// TIA Portal V18 export
// export: Created 2026-06-06T00:00:00Z, ExportSetting WithDefaults
VAR_GLOBAL   // PLC tag table "AI_Tags"
   AI_Nut_Khoi_Dong AT %I0.0 : Bool;   // Nút khởi động vật lý
   AI_Nut_Khoi_Dong_HMI AT %M110.0 : Bool;   // Tín hiệu mô phỏng/HMI song song cho Nút khởi động vật lý
   AI_Nut_Khoi_Dong_HMI_Gated AT %M320.0 : Bool;   // Tín hiệu HMI đã qua xử lý chế độ cho Nút khởi động vật lý
   AI_Nut_Khoi_Dong_Eff AT %M320.1 : Bool;   // Tín hiệu thực tế/mô phỏng hiệu dụng cho Nút khởi động vật lý
   AI_Nut_Dung AT %I0.1 : Bool;   // Nút dừng vật lý
   AI_Nut_Dung_HMI AT %M110.1 : Bool;   // Tín hiệu mô phỏng/HMI song song cho Nút dừng vật lý
   AI_Nut_Dung_HMI_Gated AT %M320.2 : Bool;   // Tín hiệu HMI đã qua xử lý chế độ cho Nút dừng vật lý
   AI_Nut_Dung_Eff AT %M320.3 : Bool;   // Tín hiệu thực tế/mô phỏng hiệu dụng cho Nút dừng vật lý
   AI_Nut_Reset AT %I0.2 : Bool;   // Nút reset lỗi vật lý
   AI_Nut_Reset_HMI AT %M110.2 : Bool;   // Tín hiệu mô phỏng/HMI song song cho Nút reset lỗi vật lý
   AI_Nut_Reset_HMI_Gated AT %M320.4 : Bool;   // Tín hiệu HMI đã qua xử lý chế độ cho Nút reset lỗi vật lý
   AI_Nut_Reset_Eff AT %M320.5 : Bool;   // Tín hiệu thực tế/mô phỏng hiệu dụng cho Nút reset lỗi vật lý
   AI_Nut_EStop AT %I0.3 : Bool;   // Nút dừng khẩn vật lý
   AI_Nut_EStop_HMI AT %M110.3 : Bool;   // Tín hiệu mô phỏng/HMI song song cho Nút dừng khẩn vật lý
   AI_Nut_EStop_HMI_Gated AT %M320.6 : Bool;   // Tín hiệu HMI đã qua xử lý chế độ cho Nút dừng khẩn vật lý
   AI_Nut_EStop_Eff AT %M320.7 : Bool;   // Tín hiệu thực tế/mô phỏng hiệu dụng cho Nút dừng khẩn vật lý
   AI_FT3200_Bon1 AT %ID100 : Real;   // Cảm biến lưu lượng nước dosing vào Bồn 1
   AI_FT3200_Bon1_HMI AT %MD700 : Real;   // Giá trị mô phỏng/HMI song song cho Cảm biến lưu lượng nước dosing vào Bồn 1
   AI_FT3200_Bon1_Use_HMI AT %M420.0 : Bool;   // Chọn chế độ mô phỏng HMI cho Cảm biến lưu lượng nước dosing vào Bồn 1
   AI_FT3200_Bon1_Sim_Req AT %M321.0 : Bool;   // Yêu cầu mô phỏng cảm biến cho Cảm biến lưu lượng nước dosing vào Bồn 1
   AI_FT3200_Bon1_Sim_Active AT %M321.1 : Bool;   // Mô phỏng cảm biến đang hoạt động cho Cảm biến lưu lượng nước dosing vào Bồn 1
   AI_FT3200_Bon1_Eff AT %MD704 : Real;   // Giá trị thực tế/mô phỏng hiệu dụng cho Cảm biến lưu lượng nước dosing vào Bồn 1
   AI_FQ3200_Bon1 AT %ID104 : Real;   // Bộ đếm lưu lượng tích lũy Bồn 1
   AI_FQ3200_Bon1_HMI AT %MD708 : Real;   // Giá trị mô phỏng/HMI song song cho Bộ đếm lưu lượng tích lũy Bồn 1
   AI_FQ3200_Bon1_Use_HMI AT %M420.1 : Bool;   // Chọn chế độ mô phỏng HMI cho Bộ đếm lưu lượng tích lũy Bồn 1
   AI_FQ3200_Bon1_Sim_Req AT %M321.2 : Bool;   // Yêu cầu mô phỏng cảm biến cho Bộ đếm lưu lượng tích lũy Bồn 1
   AI_FQ3200_Bon1_Sim_Active AT %M321.3 : Bool;   // Mô phỏng cảm biến đang hoạt động cho Bộ đếm lưu lượng tích lũy Bồn 1
   AI_FQ3200_Bon1_Eff AT %MD712 : Real;   // Giá trị thực tế/mô phỏng hiệu dụng cho Bộ đếm lưu lượng tích lũy Bồn 1
   AI_LS3202_Bon1_Cao AT %I0.4 : Bool;   // Cảm biến mức cao Bồn 1
   AI_LS3202_Bon1_Cao_HMI AT %M110.4 : Bool;   // Tín hiệu mô phỏng/HMI song song cho Cảm biến mức cao Bồn 1
   AI_LS3202_Bon1_Cao_HMI_Gated AT %M321.4 : Bool;   // Tín hiệu HMI đã qua xử lý chế độ cho Cảm biến mức cao Bồn 1
   AI_LS3202_Bon1_Cao_Eff AT %M321.5 : Bool;   // Tín hiệu thực tế/mô phỏng hiệu dụng cho Cảm biến mức cao Bồn 1
   AI_LT3203_Bon1 AT %ID108 : Real;   // Cảm biến mức liên tục Bồn 1
   AI_LT3203_Bon1_HMI AT %MD716 : Real;   // Giá trị mô phỏng/HMI song song cho Cảm biến mức liên tục Bồn 1
   AI_LT3203_Bon1_Use_HMI AT %M420.2 : Bool;   // Chọn chế độ mô phỏng HMI cho Cảm biến mức liên tục Bồn 1
   AI_LT3203_Bon1_Sim_Req AT %M321.6 : Bool;   // Yêu cầu mô phỏng cảm biến cho Cảm biến mức liên tục Bồn 1
   AI_LT3203_Bon1_Sim_Active AT %M321.7 : Bool;   // Mô phỏng cảm biến đang hoạt động cho Cảm biến mức liên tục Bồn 1
   AI_LT3203_Bon1_Eff AT %MD720 : Real;   // Giá trị thực tế/mô phỏng hiệu dụng cho Cảm biến mức liên tục Bồn 1
   AI_TT3204_Bon1 AT %ID112 : Real;   // Cảm biến nhiệt độ Bồn 1
   AI_TT3204_Bon1_HMI AT %MD724 : Real;   // Giá trị mô phỏng/HMI song song cho Cảm biến nhiệt độ Bồn 1
   AI_TT3204_Bon1_Use_HMI AT %M420.3 : Bool;   // Chọn chế độ mô phỏng HMI cho Cảm biến nhiệt độ Bồn 1
   AI_TT3204_Bon1_Sim_Req AT %M322.0 : Bool;   // Yêu cầu mô phỏng cảm biến cho Cảm biến nhiệt độ Bồn 1
   AI_TT3204_Bon1_Sim_Active AT %M322.1 : Bool;   // Mô phỏng cảm biến đang hoạt động cho Cảm biến nhiệt độ Bồn 1
   AI_TT3204_Bon1_Eff AT %MD728 : Real;   // Giá trị thực tế/mô phỏng hiệu dụng cho Cảm biến nhiệt độ Bồn 1
   AI_FT3205_Bon2 AT %ID116 : Real;   // Cảm biến lưu lượng nước dosing vào Bồn 2
   AI_FT3205_Bon2_HMI AT %MD732 : Real;   // Giá trị mô phỏng/HMI song song cho Cảm biến lưu lượng nước dosing vào Bồn 2
   AI_FT3205_Bon2_Use_HMI AT %M420.4 : Bool;   // Chọn chế độ mô phỏng HMI cho Cảm biến lưu lượng nước dosing vào Bồn 2
   AI_FT3205_Bon2_Sim_Req AT %M322.2 : Bool;   // Yêu cầu mô phỏng cảm biến cho Cảm biến lưu lượng nước dosing vào Bồn 2
   AI_FT3205_Bon2_Sim_Active AT %M322.3 : Bool;   // Mô phỏng cảm biến đang hoạt động cho Cảm biến lưu lượng nước dosing vào Bồn 2
   AI_FT3205_Bon2_Eff AT %MD736 : Real;   // Giá trị thực tế/mô phỏng hiệu dụng cho Cảm biến lưu lượng nước dosing vào Bồn 2
   AI_FQ3205_Bon2 AT %ID120 : Real;   // Bộ đếm lưu lượng tích lũy Bồn 2
   AI_FQ3205_Bon2_HMI AT %MD740 : Real;   // Giá trị mô phỏng/HMI song song cho Bộ đếm lưu lượng tích lũy Bồn 2
   AI_FQ3205_Bon2_Use_HMI AT %M420.5 : Bool;   // Chọn chế độ mô phỏng HMI cho Bộ đếm lưu lượng tích lũy Bồn 2
   AI_FQ3205_Bon2_Sim_Req AT %M322.4 : Bool;   // Yêu cầu mô phỏng cảm biến cho Bộ đếm lưu lượng tích lũy Bồn 2
   AI_FQ3205_Bon2_Sim_Active AT %M322.5 : Bool;   // Mô phỏng cảm biến đang hoạt động cho Bộ đếm lưu lượng tích lũy Bồn 2
   AI_FQ3205_Bon2_Eff AT %MD744 : Real;   // Giá trị thực tế/mô phỏng hiệu dụng cho Bộ đếm lưu lượng tích lũy Bồn 2
   AI_LT3209_Bon2 AT %ID124 : Real;   // Cảm biến mức liên tục Bồn 2
   AI_LT3209_Bon2_HMI AT %MD748 : Real;   // Giá trị mô phỏng/HMI song song cho Cảm biến mức liên tục Bồn 2
   AI_LT3209_Bon2_Use_HMI AT %M420.6 : Bool;   // Chọn chế độ mô phỏng HMI cho Cảm biến mức liên tục Bồn 2
   AI_LT3209_Bon2_Sim_Req AT %M322.6 : Bool;   // Yêu cầu mô phỏng cảm biến cho Cảm biến mức liên tục Bồn 2
   AI_LT3209_Bon2_Sim_Active AT %M322.7 : Bool;   // Mô phỏng cảm biến đang hoạt động cho Cảm biến mức liên tục Bồn 2
   AI_LT3209_Bon2_Eff AT %MD752 : Real;   // Giá trị thực tế/mô phỏng hiệu dụng cho Cảm biến mức liên tục Bồn 2
   AI_TT3208_Bon2 AT %ID128 : Real;   // Cảm biến nhiệt độ Bồn 2
   AI_TT3208_Bon2_HMI AT %MD756 : Real;   // Giá trị mô phỏng/HMI song song cho Cảm biến nhiệt độ Bồn 2
   AI_TT3208_Bon2_Use_HMI AT %M420.7 : Bool;   // Chọn chế độ mô phỏng HMI cho Cảm biến nhiệt độ Bồn 2
   AI_TT3208_Bon2_Sim_Req AT %M323.0 : Bool;   // Yêu cầu mô phỏng cảm biến cho Cảm biến nhiệt độ Bồn 2
   AI_TT3208_Bon2_Sim_Active AT %M323.1 : Bool;   // Mô phỏng cảm biến đang hoạt động cho Cảm biến nhiệt độ Bồn 2
   AI_TT3208_Bon2_Eff AT %MD760 : Real;   // Giá trị thực tế/mô phỏng hiệu dụng cho Cảm biến nhiệt độ Bồn 2
   AI_V3230_Nuoc_Bon1 AT %Q0.0 : Bool;   // Van on/off cấp nước Bồn 1
   AI_V3230_Nuoc_Bon1_M AT %M220.0 : Bool;   // Tag gương phản hồi HMI cho Van on/off cấp nước Bồn 1
   AI_CV3201_Nuoc_Bon1 AT %QD100 : Real;   // Van tuyến tính cấp nước Bồn 1
   AI_CV3201_Nuoc_Bon1_M AT %MD1200 : Real;   // Tag gương phản hồi HMI cho Van tuyến tính cấp nước Bồn 1
   AI_AGTR3260_Khuay_Bon1 AT %Q0.1 : Bool;   // Động cơ khuấy Bồn 1
   AI_AGTR3260_Khuay_Bon1_M AT %M220.1 : Bool;   // Tag gương phản hồi HMI cho Động cơ khuấy Bồn 1
   AI_AGTR3260_Toc_Do_AO AT %QD104 : Real;   // Tín hiệu tốc độ khuấy Bồn 1
   AI_AGTR3260_Toc_Do_AO_M AT %MD1204 : Real;   // Tag gương phản hồi HMI cho Tín hiệu tốc độ khuấy Bồn 1
   AI_V3232_Xa_Bon1 AT %Q0.2 : Bool;   // Van xả đáy Bồn 1 số 1
   AI_V3232_Xa_Bon1_M AT %M220.2 : Bool;   // Tag gương phản hồi HMI cho Van xả đáy Bồn 1 số 1
   AI_V3233_Xa_Bon1 AT %Q0.3 : Bool;   // Van xả đáy Bồn 1 số 2
   AI_V3233_Xa_Bon1_M AT %M220.3 : Bool;   // Tag gương phản hồi HMI cho Van xả đáy Bồn 1 số 2
   AI_V3234_Xa_Bon1 AT %Q0.4 : Bool;   // Van xả đáy Bồn 1 số 3
   AI_V3234_Xa_Bon1_M AT %M220.4 : Bool;   // Tag gương phản hồi HMI cho Van xả đáy Bồn 1 số 3
   AI_V3235_Nuoc_Bon2 AT %Q0.5 : Bool;   // Van on/off cấp nước Bồn 2
   AI_V3235_Nuoc_Bon2_M AT %M220.5 : Bool;   // Tag gương phản hồi HMI cho Van on/off cấp nước Bồn 2
   AI_CV3206_Hoi_Bon2 AT %QD108 : Real;   // Van hơi/nhiệt Bồn 2 ở chế độ cho phép
   AI_CV3206_Hoi_Bon2_M AT %MD1208 : Real;   // Tag gương phản hồi HMI cho Van hơi/nhiệt Bồn 2 ở chế độ cho phép
   AI_VFD_Bon2_Run AT %Q0.6 : Bool;   // Lệnh chạy VFD động cơ Bồn 2
   AI_VFD_Bon2_Run_M AT %M220.6 : Bool;   // Tag gương phản hồi HMI cho Lệnh chạy VFD động cơ Bồn 2
   AI_VFD_Bon2_Dao_Chieu AT %Q0.7 : Bool;   // Lệnh đảo chiều VFD động cơ Bồn 2
   AI_VFD_Bon2_Dao_Chieu_M AT %M220.7 : Bool;   // Tag gương phản hồi HMI cho Lệnh đảo chiều VFD động cơ Bồn 2
   AI_VFD_Bon2_Toc_Do_AO AT %QD112 : Real;   // Tốc độ đặt VFD Bồn 2 từ HMI setpoint
   AI_VFD_Bon2_Toc_Do_AO_M AT %MD1212 : Real;   // Tag gương phản hồi HMI cho Tốc độ đặt VFD Bồn 2 từ HMI setpoint
   AI_V3237_Xa_Bon2 AT %Q1.0 : Bool;   // Van xả đáy Bồn 2 số 1
   AI_V3237_Xa_Bon2_M AT %M221.0 : Bool;   // Tag gương phản hồi HMI cho Van xả đáy Bồn 2 số 1
   AI_V3238_Xa_Bon2 AT %Q1.1 : Bool;   // Van xả đáy Bồn 2 số 2
   AI_V3238_Xa_Bon2_M AT %M221.1 : Bool;   // Tag gương phản hồi HMI cho Van xả đáy Bồn 2 số 2
   AI_V3239_Xa_Bon2 AT %Q1.2 : Bool;   // Van xả đáy Bồn 2 số 3
   AI_V3239_Xa_Bon2_M AT %M221.2 : Bool;   // Tag gương phản hồi HMI cho Van xả đáy Bồn 2 số 3
   AI_Pump3264_Chuyen_Nhanh1 AT %Q1.3 : Bool;   // Bơm chuyển dung dịch Nhánh 1 xuống bồn chứa
   AI_Pump3264_Chuyen_Nhanh1_M AT %M221.3 : Bool;   // Tag gương phản hồi HMI cho Bơm chuyển dung dịch Nhánh 1 xuống bồn chứa
   AI_LT3302_BonChua1 AT %ID164 : Real;   // Cảm biến mức liên tục Bồn chứa 01
   AI_LT3302_BonChua1_HMI AT %MD828 : Real;   // Giá trị mô phỏng/HMI song song cho Cảm biến mức liên tục Bồn chứa 01
   AI_LT3302_BonChua1_Use_HMI AT %M422.0 : Bool;   // Chọn chế độ mô phỏng HMI cho Cảm biến mức liên tục Bồn chứa 01
   AI_LT3302_BonChua1_Sim_Req AT %M325.4 : Bool;   // Yêu cầu mô phỏng cảm biến cho Cảm biến mức liên tục Bồn chứa 01
   AI_LT3302_BonChua1_Sim_Active AT %M325.5 : Bool;   // Mô phỏng cảm biến đang hoạt động cho Cảm biến mức liên tục Bồn chứa 01
   AI_LT3302_BonChua1_Eff AT %MD832 : Real;   // Giá trị thực tế/mô phỏng hiệu dụng cho Cảm biến mức liên tục Bồn chứa 01
   AI_TT3301_BonChua1 AT %ID168 : Real;   // Cảm biến nhiệt độ Bồn chứa 01
   AI_TT3301_BonChua1_HMI AT %MD836 : Real;   // Giá trị mô phỏng/HMI song song cho Cảm biến nhiệt độ Bồn chứa 01
   AI_TT3301_BonChua1_Use_HMI AT %M422.1 : Bool;   // Chọn chế độ mô phỏng HMI cho Cảm biến nhiệt độ Bồn chứa 01
   AI_TT3301_BonChua1_Sim_Req AT %M325.6 : Bool;   // Yêu cầu mô phỏng cảm biến cho Cảm biến nhiệt độ Bồn chứa 01
   AI_TT3301_BonChua1_Sim_Active AT %M325.7 : Bool;   // Mô phỏng cảm biến đang hoạt động cho Cảm biến nhiệt độ Bồn chứa 01
   AI_TT3301_BonChua1_Eff AT %MD840 : Real;   // Giá trị thực tế/mô phỏng hiệu dụng cho Cảm biến nhiệt độ Bồn chứa 01
   AI_TT3303_TraoDoiNhiet AT %ID172 : Real;   // Cảm biến nhiệt độ bộ trao đổi nhiệt
   AI_TT3303_TraoDoiNhiet_HMI AT %MD844 : Real;   // Giá trị mô phỏng/HMI song song cho Cảm biến nhiệt độ bộ trao đổi nhiệt
   AI_TT3303_TraoDoiNhiet_Use_HMI AT %M422.2 : Bool;   // Chọn chế độ mô phỏng HMI cho Cảm biến nhiệt độ bộ trao đổi nhiệt
   AI_TT3303_TraoDoiNhiet_Sim_Req AT %M326.0 : Bool;   // Yêu cầu mô phỏng cảm biến cho Cảm biến nhiệt độ bộ trao đổi nhiệt
   AI_TT3303_TraoDoiNhiet_Sim_Active AT %M326.1 : Bool;   // Mô phỏng cảm biến đang hoạt động cho Cảm biến nhiệt độ bộ trao đổi nhiệt
   AI_TT3303_TraoDoiNhiet_Eff AT %MD848 : Real;   // Giá trị thực tế/mô phỏng hiệu dụng cho Cảm biến nhiệt độ bộ trao đổi nhiệt
   AI_LT3307_BonChua2 AT %ID176 : Real;   // Cảm biến mức liên tục Bồn chứa 02
   AI_LT3307_BonChua2_HMI AT %MD852 : Real;   // Giá trị mô phỏng/HMI song song cho Cảm biến mức liên tục Bồn chứa 02
   AI_LT3307_BonChua2_Use_HMI AT %M422.3 : Bool;   // Chọn chế độ mô phỏng HMI cho Cảm biến mức liên tục Bồn chứa 02
   AI_LT3307_BonChua2_Sim_Req AT %M326.2 : Bool;   // Yêu cầu mô phỏng cảm biến cho Cảm biến mức liên tục Bồn chứa 02
   AI_LT3307_BonChua2_Sim_Active AT %M326.3 : Bool;   // Mô phỏng cảm biến đang hoạt động cho Cảm biến mức liên tục Bồn chứa 02
   AI_LT3307_BonChua2_Eff AT %MD856 : Real;   // Giá trị thực tế/mô phỏng hiệu dụng cho Cảm biến mức liên tục Bồn chứa 02
   AI_TT3306_BonChua2 AT %ID180 : Real;   // Cảm biến nhiệt độ Bồn chứa 02
   AI_TT3306_BonChua2_HMI AT %MD860 : Real;   // Giá trị mô phỏng/HMI song song cho Cảm biến nhiệt độ Bồn chứa 02
   AI_TT3306_BonChua2_Use_HMI AT %M422.4 : Bool;   // Chọn chế độ mô phỏng HMI cho Cảm biến nhiệt độ Bồn chứa 02
   AI_TT3306_BonChua2_Sim_Req AT %M326.4 : Bool;   // Yêu cầu mô phỏng cảm biến cho Cảm biến nhiệt độ Bồn chứa 02
   AI_TT3306_BonChua2_Sim_Active AT %M326.5 : Bool;   // Mô phỏng cảm biến đang hoạt động cho Cảm biến nhiệt độ Bồn chứa 02
   AI_TT3306_BonChua2_Eff AT %MD864 : Real;   // Giá trị thực tế/mô phỏng hiệu dụng cho Cảm biến nhiệt độ Bồn chứa 02
   AI_PI3308_Truoc_Filter AT %ID184 : Real;   // Cảm biến áp suất trước màng lọc
   AI_PI3308_Truoc_Filter_HMI AT %MD868 : Real;   // Giá trị mô phỏng/HMI song song cho Cảm biến áp suất trước màng lọc
   AI_PI3308_Truoc_Filter_Use_HMI AT %M422.5 : Bool;   // Chọn chế độ mô phỏng HMI cho Cảm biến áp suất trước màng lọc
   AI_PI3308_Truoc_Filter_Sim_Req AT %M326.6 : Bool;   // Yêu cầu mô phỏng cảm biến cho Cảm biến áp suất trước màng lọc
   AI_PI3308_Truoc_Filter_Sim_Active AT %M326.7 : Bool;   // Mô phỏng cảm biến đang hoạt động cho Cảm biến áp suất trước màng lọc
   AI_PI3308_Truoc_Filter_Eff AT %MD872 : Real;   // Giá trị thực tế/mô phỏng hiệu dụng cho Cảm biến áp suất trước màng lọc
   AI_FT3309_Xa_Thanh_Pham AT %ID188 : Real;   // Cảm biến lưu lượng xả thành phẩm
   AI_FT3309_Xa_Thanh_Pham_HMI AT %MD876 : Real;   // Giá trị mô phỏng/HMI song song cho Cảm biến lưu lượng xả thành phẩm
   AI_FT3309_Xa_Thanh_Pham_Use_HMI AT %M422.6 : Bool;   // Chọn chế độ mô phỏng HMI cho Cảm biến lưu lượng xả thành phẩm
   AI_FT3309_Xa_Thanh_Pham_Sim_Req AT %M327.0 : Bool;   // Yêu cầu mô phỏng cảm biến cho Cảm biến lưu lượng xả thành phẩm
   AI_FT3309_Xa_Thanh_Pham_Sim_Active AT %M327.1 : Bool;   // Mô phỏng cảm biến đang hoạt động cho Cảm biến lưu lượng xả thành phẩm
   AI_FT3309_Xa_Thanh_Pham_Eff AT %MD880 : Real;   // Giá trị thực tế/mô phỏng hiệu dụng cho Cảm biến lưu lượng xả thành phẩm
   AI_LSH3310_Pheu_Cao AT %I0.6 : Bool;   // Cảm biến mức cao phễu chiết rót
   AI_LSH3310_Pheu_Cao_HMI AT %M110.6 : Bool;   // Tín hiệu mô phỏng/HMI song song cho Cảm biến mức cao phễu chiết rót
   AI_LSH3310_Pheu_Cao_HMI_Gated AT %M327.2 : Bool;   // Tín hiệu HMI đã qua xử lý chế độ cho Cảm biến mức cao phễu chiết rót
   AI_LSH3310_Pheu_Cao_Eff AT %M327.3 : Bool;   // Tín hiệu thực tế/mô phỏng hiệu dụng cho Cảm biến mức cao phễu chiết rót
   AI_LSL3311_Pheu_Thap AT %I0.7 : Bool;   // Cảm biến mức thấp phễu chiết rót
   AI_LSL3311_Pheu_Thap_HMI AT %M110.7 : Bool;   // Tín hiệu mô phỏng/HMI song song cho Cảm biến mức thấp phễu chiết rót
   AI_LSL3311_Pheu_Thap_HMI_Gated AT %M327.4 : Bool;   // Tín hiệu HMI đã qua xử lý chế độ cho Cảm biến mức thấp phễu chiết rót
   AI_LSL3311_Pheu_Thap_Eff AT %M327.5 : Bool;   // Tín hiệu thực tế/mô phỏng hiệu dụng cho Cảm biến mức thấp phễu chiết rót
   AI_V3331_Xa_BonChua1 AT %Q3.0 : Bool;   // Van xả đáy Bồn chứa 01 số 1
   AI_V3331_Xa_BonChua1_M AT %M223.0 : Bool;   // Tag gương phản hồi HMI cho Van xả đáy Bồn chứa 01 số 1
   AI_V3332_Xa_BonChua1 AT %Q3.1 : Bool;   // Van xả đáy Bồn chứa 01 số 2
   AI_V3332_Xa_BonChua1_M AT %M223.1 : Bool;   // Tag gương phản hồi HMI cho Van xả đáy Bồn chứa 01 số 2
   AI_Pump3361_LuanChuyen_BonChua1 AT %Q3.2 : Bool;   // Bơm luân chuyển Bồn chứa 01
   AI_Pump3361_LuanChuyen_BonChua1_M AT %M223.2 : Bool;   // Tag gương phản hồi HMI cho Bơm luân chuyển Bồn chứa 01
   AI_Pump3362_Xa_BonChua1 AT %Q3.3 : Bool;   // Bơm xả Bồn chứa 01
   AI_Pump3362_Xa_BonChua1_M AT %M223.3 : Bool;   // Tag gương phản hồi HMI cho Bơm xả Bồn chứa 01
   AI_V3333_DieuHuong_BonChua1 AT %Q3.4 : Bool;   // Van điều hướng Bồn chứa 01 số 1
   AI_V3333_DieuHuong_BonChua1_M AT %M223.4 : Bool;   // Tag gương phản hồi HMI cho Van điều hướng Bồn chứa 01 số 1
   AI_V3334_DieuHuong_BonChua1 AT %Q3.5 : Bool;   // Van điều hướng Bồn chứa 01 số 2
   AI_V3334_DieuHuong_BonChua1_M AT %M223.5 : Bool;   // Tag gương phản hồi HMI cho Van điều hướng Bồn chứa 01 số 2
   AI_V3335_DieuHuong_BonChua1 AT %Q3.6 : Bool;   // Van điều hướng Bồn chứa 01 số 3
   AI_V3335_DieuHuong_BonChua1_M AT %M223.6 : Bool;   // Tag gương phản hồi HMI cho Van điều hướng Bồn chứa 01 số 3
   AI_CV3304_Nuoc_Lam_Mat AT %QD132 : Real;   // Van tuyến tính nước làm mát
   AI_CV3304_Nuoc_Lam_Mat_M AT %MD1232 : Real;   // Tag gương phản hồi HMI cho Van tuyến tính nước làm mát
   AI_V3338_Xa_BonChua2 AT %Q3.7 : Bool;   // Van xả đáy Bồn chứa 02 số 1
   AI_V3338_Xa_BonChua2_M AT %M223.7 : Bool;   // Tag gương phản hồi HMI cho Van xả đáy Bồn chứa 02 số 1
   AI_V3339_Xa_BonChua2 AT %Q4.0 : Bool;   // Van xả đáy Bồn chứa 02 số 2
   AI_V3339_Xa_BonChua2_M AT %M224.0 : Bool;   // Tag gương phản hồi HMI cho Van xả đáy Bồn chứa 02 số 2
   AI_Pump3364_Filter AT %Q4.1 : Bool;   // Bơm qua màng lọc CCP số 1
   AI_Pump3364_Filter_M AT %M224.1 : Bool;   // Tag gương phản hồi HMI cho Bơm qua màng lọc CCP số 1
   AI_Pump3365_Filter AT %Q4.2 : Bool;   // Bơm qua màng lọc CCP số 2
   AI_Pump3365_Filter_M AT %M224.2 : Bool;   // Tag gương phản hồi HMI cho Bơm qua màng lọc CCP số 2
   AI_V3340_Duong_Filter AT %Q4.3 : Bool;   // Van đường ống Filter số 1
   AI_V3340_Duong_Filter_M AT %M224.3 : Bool;   // Tag gương phản hồi HMI cho Van đường ống Filter số 1
   AI_V3341_Duong_Filter AT %Q4.4 : Bool;   // Van đường ống Filter số 2
   AI_V3341_Duong_Filter_M AT %M224.4 : Bool;   // Tag gương phản hồi HMI cho Van đường ống Filter số 2
   AI_CV_Filler_Cap_Dich AT %QD136 : Real;   // Van tuyến tính cấp dịch xuống phễu chiết rót
   AI_CV_Filler_Cap_Dich_M AT %MD1236 : Real;   // Tag gương phản hồi HMI cho Van tuyến tính cấp dịch xuống phễu chiết rót
   AI_Coi_Bao_Dong AT %Q4.5 : Bool;   // Còi báo động chung
   AI_Coi_Bao_Dong_M AT %M224.5 : Bool;   // Tag gương phản hồi HMI cho Còi báo động chung
   AI_HMI_Operator_Login AT %M422.7 : Bool;   // Đăng nhập quyền Operator
   AI_HMI_Engineer_Login AT %M423.0 : Bool;   // Đăng nhập quyền Engineer
   AI_HMI_Admin_Login AT %M423.1 : Bool;   // Đăng nhập quyền Admin
   AI_HMI_Che_Do_Manual AT %M423.2 : Bool;   // Cho phép điều khiển tay từng thiết bị
   AI_HMI_Ack_Alarm AT %M423.3 : Bool;   // Xác nhận cảnh báo
   AI_HMI_Reset_Alarm AT %M423.4 : Bool;   // Reset alarm bằng HMI
   AI_Gia_Lap_Mat_Ket_Noi_HMI AT %M423.5 : Bool;   // Nút giả lập mất kết nối PLC
   AI_HMI_User_Level AT %MW520 : Int;   // Mức quyền hiện tại: 1 Operator, 2 Engineer, 3 Admin
   AI_HMI_Cho_Phep_Sua_Thong_So AT %M327.6 : Bool;   // Cờ cho phép sửa công thức và PID
   AI_HMI_Alarm_Status AT %MW522 : Int;   // Mã cảnh báo tổng hợp cho WinCC TextList
   AI_HMI_AnToan_Status AT %MW524 : Int;   // Mã chẩn đoán an toàn ưu tiên
   AI_PLC1_Auto_Enable AT %M327.7 : Bool;   // Cho phép chạy Auto Nhánh 1 Bồn 1-2
   AI_PLC1_EStop_Latch AT %M328.0 : Bool;   // Chốt dừng khẩn HMI/SCADA Nhánh 1 Bồn 1-2
   AI_PLC1_Loi_Tong AT %M328.1 : Bool;   // Lỗi tổng khóa Auto Nhánh 1 Bồn 1-2
   AI_PLC1_Loi_Dry_Run AT %M328.2 : Bool;   // Lỗi chạy khô bơm Nhánh 1 Bồn 1-2
   AI_PLC1_Loi_Dosing AT %M328.3 : Bool;   // Lỗi quá thời gian dosing Nhánh 1 Bồn 1-2
   AI_PLC1_Loi_Truyen_Thong AT %M328.4 : Bool;   // Lỗi truyền thông mô phỏng Nhánh 1 Bồn 1-2
   AI_PLC1_State AT %MW526 : Int;   // Mã bước chu trình Nhánh 1 Bồn 1-2
   AI_PLC1_Step_Bon1_Dosing AT %M329.3 : Bool;   // Bồn 1 đang dosing nước
   AI_PLC1_Step_Bon1_Tip AT %M329.4 : Bool;   // Bồn 1 đang mô phỏng tip cốt tương Nhật Bản
   AI_PLC1_Step_Bon1_Khuay AT %M329.5 : Bool;   // Bồn 1 đang khuấy ban đầu
   AI_PLC1_Step_Bon1_Xa AT %M329.6 : Bool;   // Bồn 1 đang xả sang Bồn 2
   AI_PLC1_Step_Bon2_Dosing AT %M329.7 : Bool;   // Bồn 2 đang dosing bổ sung
   AI_PLC1_Step_Bon2_Tip AT %M330.0 : Bool;   // Bồn 2 đang tip phụ gia
   AI_PLC1_Step_Bon2_Khuay_Thuan AT %M330.1 : Bool;   // Bồn 2 khuấy chiều thuận
   AI_PLC1_Step_Bon2_Khuay_Nghich AT %M330.2 : Bool;   // Bồn 2 khuấy chiều ngược
   AI_PLC1_Step_Bon2_PID AT %M330.3 : Bool;   // Bồn 2 gia nhiệt PID
   AI_PLC1_Step_Bon2_Thanh_Trung AT %M330.4 : Bool;   // Bồn 2 giữ thời gian thanh trùng
   AI_PLC1_Me_Nhanh1_Hoan_Thanh AT %M330.5 : Bool;   // Nhánh 1 hoàn thành và sẵn sàng xả xuống bồn chứa
   AI_PLC1_Xa_Bon1_Xong AT %M330.6 : Bool;   // Bồn 1 đã xả hết
   AI_PLC1_Xa_Bon2_Xong AT %M330.7 : Bool;   // Bồn 2 đã xả hết
   AI_BonChua_Step_Nhan_Dich AT %M332.4 : Bool;   // Bồn chứa 01 đang nhận dịch từ nhánh hoàn thành
   AI_BonChua_Step_Giai_Nhiet AT %M332.5 : Bool;   // Bồn chứa 01 đang giải nhiệt xuống 45 độ C
   AI_BonChua_Step_Chuyen_Bon2 AT %M332.6 : Bool;   // Đang chuyển từ Bồn chứa 01 sang Bồn chứa 02
   AI_BonChua_Step_Loc_Chiet AT %M332.7 : Bool;   // Đang lọc CCP và chiết rót
   AI_BonChua_Me_Hoan_Thanh AT %M333.0 : Bool;   // Hoàn thành một mẻ sản xuất chung
   AI_BonChua_State AT %MW530 : Int;   // Mã bước cụm bồn chứa và lọc thành phẩm
   AI_BonChua_Owner_Nhanh1 AT %M333.1 : Bool;   // Mức ưu tiên Nhánh 1 sở hữu bồn chứa
   AI_BonChua_Owner_Nhanh2 AT %M333.2 : Bool;   // Mức ưu tiên Nhánh 2 sở hữu bồn chứa
   AI_PLC2_Me_Nhanh2_Hoan_Thanh_Nhan AT %M333.4 : Bool;   // Cờ PLC1 nhận trạng thái hoàn thành từ PLC2
   AI_PLC2_Me_Nhanh2_Hoan_Thanh_Nhan_HMI AT %M111.0 : Bool;   // Tín hiệu mô phỏng/HMI song song cho cờ PLC1 nhận trạng thái hoàn thành từ PLC2
   AI_PLC2_Xa_Bon4_Xong_Nhan AT %M333.5 : Bool;   // Cờ PLC1 nhận trạng thái xả xong Bồn 4 từ PLC2
   AI_Pump3265_Chuyen_Nhanh2_Cmd AT %M333.6 : Bool;   // Lệnh chạy bơm chuyển Nhánh 2 gửi sang PLC2
   AI_Pump3265_Chuyen_Nhanh2_Cmd_M AT %M224.7 : Bool;   // Tag gương phản hồi HMI cho lệnh chạy bơm chuyển Nhánh 2 gửi sang PLC2
   AI_PID_Bon4_SP_Recv AT %MD884 : Real;   // PID Bồn 4 Setpoint nhận từ PLC2
   AI_PID_Bon4_PV_Recv AT %MD888 : Real;   // PID Bồn 4 Process Value nhận từ PLC2
   AI_PID_Bon4_CV_Recv AT %MD892 : Real;   // PID Bồn 4 Control Value nhận từ PLC2
   AI_PLC2_State_Recv AT %MW532 : Int;   // Trạng thái hoạt động PLC2 nhận từ PLC2
   AI_PLC2_Loi_Tong_Recv AT %M334.0 : Bool;   // Cờ lỗi tổng PLC2 nhận từ PLC2
   AI_VFD_Bon2_iStep AT %MW60 : Int;   // Bước quét tuần tự Modbus VFD Bồn 2
   AI_VFD_Bon2_iStep_Reset AT %M335.5 : Bool;   // Cờ reset bộ đếm bước Modbus VFD Bồn 2
   AI_VFD_Bon2_Step0_Req AT %M335.6 : Bool;   // Yêu cầu bước 0 Modbus VFD Bồn 2
   AI_VFD_Bon2_Step1_Req AT %M335.7 : Bool;   // Yêu cầu bước 1 Modbus VFD Bồn 2
   AI_VFD_Bon2_Step2_Req AT %M336.0 : Bool;   // Yêu cầu bước 2 Modbus VFD Bồn 2
   AI_VFD_Bon2_Step3_Req AT %M336.1 : Bool;   // Yêu cầu bước 3 Modbus VFD Bồn 2
   AI_VFD_Bon2_MB_ControlWord AT %MW40 : Word;   // Control Word gửi VFD Bồn 2
   AI_VFD_Bon2_MB_FreqSetpoint AT %MW42 : Int;   // Frequency Setpoint gửi VFD Bồn 2
   AI_VFD_Bon2_MB_StatusWord AT %MW44 : Word;   // Status Word đọc từ VFD Bồn 2
   AI_VFD_Bon2_MB_ActualSpeed AT %MW46 : Int;   // Actual Speed đọc từ VFD Bồn 2
   AI_VFD_Bon2_MB_Error AT %M50.0 : Bool;   // Lỗi Modbus Master VFD Bồn 2
   AI_VFD_Bon2_MB_Busy AT %M50.1 : Bool;   // Modbus Master Busy VFD Bồn 2
   AI_VFD_Bon2_MB_Done AT %M50.2 : Bool;   // Modbus Master Done VFD Bồn 2
   AI_VFD_Bon2_MB_Status AT %MW52 : Word;   // Trạng thái Modbus Master VFD Bồn 2
   AI_VFD_Bon2_MBCL_Done AT %M51.0 : Bool;   // Modbus Comm Load Done VFD Bồn 2
   AI_VFD_Bon2_MBCL_Error AT %M51.1 : Bool;   // Modbus Comm Load Error VFD Bồn 2
   AI_VFD_Bon2_MBCL_Status AT %MW54 : Word;   // Trạng thái Modbus Comm Load VFD Bồn 2
   AI_VFD_Bon2_Freq_Temp AT %MD70 : Real;   // Biến tạm tần số VFD Bồn 2
   AI_VFD_Bon2_Actual_Speed_Feedback AT %MD74 : Real;   // Phản hồi tốc độ thực tế VFD Bồn 2
   AI_VFD_Bon2_Actual_Speed_Feedback_M AT %MD1240 : Real;   // Tag gương phản hồi HMI tốc độ thực tế VFD Bồn 2
   AI_Clock_1Hz AT %M100.5 : Bool;   // Clock 1Hz system memory bit
   AI_FirstScan AT %M101.0 : Bool;   // First Scan system memory bit
   AI_MB_TCP_iStep AT %MW80 : Int;   // Modbus TCP Client step
   AI_MB_TCP_REQ AT %M82.0 : Bool;   // Modbus TCP Client Request
   AI_MB_TCP_DONE AT %M82.2 : Bool;   // Modbus TCP Client Transaction Done
   AI_MB_TCP_ERROR AT %M82.3 : Bool;   // Modbus TCP Client Transaction Error
   AI_MB_TCP_BUSY AT %M82.6 : Bool;   // Modbus TCP Client Transaction Busy
   AI_MB_TCP_STATUS AT %MW84 : Word;   // Modbus TCP Client Status
   AI_MB_TCP_Mode AT %MB88 : USInt;   // Modbus TCP Client Mode
   AI_MB_TCP_DataAddr AT %MD90 : UDInt;   // Modbus TCP Client Data Address
   AI_MB_TCP_DataLen AT %MW94 : UInt;   // Modbus TCP Client Data Length
   AI_Nut_Khoi_Dong_Eff_Old AT %M83.0 : Bool;   // Old value of Start button
   AI_Nut_Khoi_Dong_Eff_Edge AT %M83.6 : Bool;   // Start command edge detected
   AI_Nut_Dung_Eff_Old AT %M83.1 : Bool;   // Old value of Stop button
   AI_Nut_Dung_Eff_Edge AT %M83.7 : Bool;   // Stop command edge detected
   AI_Nut_Reset_Eff_Old AT %M83.2 : Bool;   // Old value of Reset button
   AI_Nut_Reset_Eff_Edge AT %M84.0 : Bool;   // Reset command edge detected
   AI_Nut_EStop_Eff_Old AT %M83.3 : Bool;   // Old value of EStop button
   AI_Nut_EStop_Eff_Edge AT %M84.1 : Bool;   // EStop command edge detected
   AI_Pump3265_Chuyen_Nhanh2_Cmd_Old AT %M83.4 : Bool;   // Old value of Transfer command
   AI_Pump3265_Chuyen_Nhanh2_Cmd_Edge AT %M84.2 : Bool;   // Transfer command edge detected
   AI_PLC1_Load_Default_Cmd_Old AT %M83.5 : Bool;   // Old value of Load Recipe command
   AI_PLC1_Load_Default_Cmd_Edge AT %M84.3 : Bool;   // Load Recipe command edge detected
   AI_MB_TCP_Any_Cmd_Edge AT %M84.4 : Bool;   // Any handshake command edge detected
   AI_PLC1_Tip_Bon1_Xong_HMI AT %M423.6 : Bool;   // Nút mô phỏng tip Bồn 1 đã hoàn tất
   AI_PLC1_Khuay_Bon1_Xong_HMI AT %M423.7 : Bool;   // Nút mô phỏng hết thời gian khuấy Bồn 1
   AI_PLC1_Tip_Bon2_Xong_HMI AT %M424.0 : Bool;   // Nút mô phỏng tip Bồn 2 đã hoàn tất
   AI_PLC1_Khuay_Thuan_Bon2_Xong_HMI AT %M424.1 : Bool;   // Nút mô phỏng hết thời gian khuấy thuận Bồn 2
   AI_PLC1_Khuay_Nghich_Bon2_Xong_HMI AT %M424.2 : Bool;   // Nút mô phỏng hết thời gian khuấy ngược Bồn 2
   AI_PLC1_Thanh_Trung_Bon2_Xong_HMI AT %M424.3 : Bool;   // Nút mô phỏng hết thời gian thanh trùng Bồn 2
   AI_PLC2_Tip_Bon3_Xong_HMI AT %M424.4 : Bool;   // Nút mô phỏng tip Bồn 3 đã hoàn tất
   AI_PLC2_Khuay_Bon3_Xong_HMI AT %M424.5 : Bool;   // Nút mô phỏng hết thời gian khuấy Bồn 3
   AI_PLC2_Tip_Bon4_Xong_HMI AT %M424.6 : Bool;   // Nút mô phỏng tip Bồn 4 đã hoàn tất
   AI_PLC2_Khuay_Thuan_Bon4_Xong_HMI AT %M424.7 : Bool;   // Nút mô phỏng hết thời gian khuấy thuận Bồn 4
   AI_PLC2_Khuay_Nghich_Bon4_Xong_HMI AT %M425.0 : Bool;   // Nút mô phỏng hết thời gian khuấy ngược Bồn 4
   AI_PLC2_Thanh_Trung_Bon4_Xong_HMI AT %M425.1 : Bool;   // Nút mô phỏng hết thời gian thanh trùng Bồn 4
   AI_BonChua_Nhan_Dich_Xong_HMI AT %M425.2 : Bool;   // Nút mô phỏng nhận dịch vào Bồn chứa 01 xong
   AI_BonChua_Chuyen_Bon2_Xong_HMI AT %M425.3 : Bool;   // Nút mô phỏng chuyển sang Bồn chứa 02 xong
   AI_HMI_SP_PLC1_Nuoc_Bon1 AT %MD896 : Real;   // Lượng nước dosing Bồn 1
   AI_HMI_SP_PLC1_Nuoc_Bon2 AT %MD900 : Real;   // Lượng nước dosing bổ sung Bồn 2
   AI_HMI_SP_PLC1_Toc_Do_Bon1 AT %MD904 : Real;   // Tốc độ khuấy Bồn 1
   AI_HMI_SP_PLC1_Toc_Do_Bon2_Main AT %MD908 : Real;   // Tốc độ khuấy chính Bồn 2
   AI_HMI_SP_PLC1_Nhiet_Do_Bon2 AT %MD912 : Real;   // Setpoint nhiệt/PID Bồn 2
   AI_HMI_SP_PLC2_Nuoc_Bon3 AT %MD916 : Real;   // Lượng nước dosing Bồn 3
   AI_HMI_SP_PLC2_Nuoc_Bon4 AT %MD920 : Real;   // Lượng nước dosing bổ sung Bồn 4
   AI_HMI_SP_PLC2_Toc_Do_Bon3 AT %MD924 : Real;   // Tốc độ khuấy Bồn 3
   AI_HMI_SP_PLC2_Toc_Do_Bon4_Main AT %MD928 : Real;   // Tốc độ khuấy chính Bồn 4
   AI_HMI_SP_PLC2_Nhiet_Do_Bon4 AT %MD932 : Real;   // Setpoint nhiệt/PID mô phỏng Bồn 4
   AI_HMI_SP_BonChua1_Nhiet_Giai_Nhiet AT %MD936 : Real;   // Nhiệt độ giải nhiệt đích Bồn chứa 01
   AI_HMI_SP_Loc_Ap_Suat_Max AT %MD940 : Real;   // Ngưỡng áp suất cao trước màng lọc
   AI_HMI_SP_Time_Khuay_Bon1 AT %MD944 : Time;   // Thời gian khuấy Bồn 1
   AI_HMI_SP_Time_Khuay_Bon3 AT %MD948 : Time;   // Thời gian khuấy Bồn 3
   AI_HMI_SP_Time_Fwd AT %MD952 : Time;   // Thời gian khuấy chiều thuận
   AI_HMI_SP_Time_Rev AT %MD956 : Time;   // Thời gian khuấy chiều ngược
   AI_HMI_SP_Time_Sterilize AT %MD960 : Time;   // Thời gian giữ nhiệt thanh trùng
   AI_PLC1_Khuay_Bon1_Xong AT %M336.2 : Bool;   // Trạng thái tự động xong khuấy Bồn 1
   AI_PLC1_Khuay_Thuan_Bon2_Xong AT %M336.3 : Bool;   // Trạng thái tự động xong khuấy thuận Bồn 2
   AI_PLC1_Khuay_Nghich_Bon2_Xong AT %M336.4 : Bool;   // Trạng thái tự động xong khuấy ngược Bồn 2
   AI_PLC1_Thanh_Trung_Bon2_Xong AT %M336.5 : Bool;   // Trạng thái tự động xong thanh trùng Bồn 2
   AI_PLC2_Khuay_Bon3_Xong AT %M336.6 : Bool;   // Trạng thái tự động xong khuấy Bồn 3
   AI_PLC2_Khuay_Thuan_Bon4_Xong AT %M336.7 : Bool;   // Trạng thái tự động xong khuấy thuận Bồn 4
   AI_PLC2_Khuay_Nghich_Bon4_Xong AT %M337.0 : Bool;   // Trạng thái tự động xong khuấy ngược Bồn 4
   AI_PLC2_Thanh_Trung_Bon4_Xong AT %M337.1 : Bool;   // Trạng thái tự động xong thanh trùng Bồn 4
   AI_PLC1_Tip_Bon1_Auto_Done AT %M337.2 : Bool;   // Trạng thái tự động xong tip Bồn 1
   AI_PLC1_Tip_Bon2_Auto_Done AT %M337.3 : Bool;   // Trạng thái tự động xong tip Bồn 2
   AI_PLC2_Tip_Bon3_Auto_Done AT %M337.4 : Bool;   // Trạng thái tự động xong tip Bồn 3
   AI_PLC2_Tip_Bon4_Auto_Done AT %M337.5 : Bool;   // Trạng thái tự động xong tip Bồn 4
   AI_PLC1_Start_Edge_Old AT %M337.6 : Bool;   // Cờ nhớ cạnh lên nút Start PLC1
   AI_PLC1_Start_Edge_Edge AT %M337.7 : Bool;   // Xung cạnh lên nút Start PLC1
   AI_PLC2_Start_Edge_Old AT %M338.0 : Bool;   // Cờ nhớ cạnh lên nút Start PLC2
   AI_PLC2_Start_Edge_Edge AT %M338.1 : Bool;   // Xung cạnh lên nút Start PLC2
   AI_PID_Bon2_Enable AT %M338.2 : Bool;   // Cho phép PID Bồn 2
   AI_PID_Bon2_ManualEnable AT %M338.3 : Bool;   // Chế độ manual PID Bồn 2
   AI_PID_Bon2_Error AT %M338.4 : Bool;   // Lỗi khối PID Bồn 2
   AI_PID_Bon2_Reset_Eff AT %M338.5 : Bool;   // Reset hiệu dụng PID Bồn 2
   AI_PID_Bon4_Enable AT %M338.6 : Bool;   // Cho phép PID mô phỏng Bồn 4
   AI_PID_Bon4_ManualEnable AT %M338.7 : Bool;   // Chế độ manual PID Bồn 4
   AI_PID_Bon4_Error AT %M339.0 : Bool;   // Lỗi khối PID Bồn 4
   AI_PID_Bon4_Reset_Eff AT %M339.1 : Bool;   // Reset hiệu dụng PID Bồn 4
   AI_PID_Bon2_ErrorBits AT %MD964 : DWord;   // Mã lỗi DWORD PID Bồn 2
   AI_PID_Bon4_ErrorBits AT %MD968 : DWord;   // Mã lỗi DWORD PID Bồn 4
   AI_PID_Bon2_SP AT %MD972 : Real;   // Setpoint đưa vào PID Bồn 2
   AI_PID_Bon2_Err AT %MD976 : Real;   // Sai lệch PID Bồn 2 = SP - PV
   AI_PID_Bon2_CV AT %MD980 : Real;   // Giá trị điều khiển PID Bồn 2
   AI_PID_Bon2_ManualValue AT %MD984 : Real;   // Giá trị manual PID Bồn 2
   AI_PID_Bon4_SP AT %MD988 : Real;   // Setpoint đưa vào PID mô phỏng Bồn 4
   AI_PID_Bon4_Err AT %MD992 : Real;   // Sai lệch PID mô phỏng Bồn 4 = SP - PV
   AI_PID_Bon4_CV AT %MD996 : Real;   // Giá trị điều khiển PID mô phỏng Bồn 4
   AI_PID_Bon4_ManualValue AT %MD1000 : Real;   // Giá trị manual PID Bồn 4
   AI_TT3219_Bon4_Sim AT %MD1004 : Real;   // Nhiệt độ mô phỏng nội bộ cho PID Bồn 4
   AI_PID_Bon2_Temp_Inc AT %MD1008 : Real;   // Mức tăng nhiệt mô phỏng Bồn 2
   AI_PID_Bon4_Tang_Nhiet_Buoc AT %MD1012 : Real;   // Mức tăng nhiệt mô phỏng mỗi chu kỳ OB31
   AI_TT3219_Bon4_Target AT %MD1016 : Real;   // Nhiệt độ đích mô phỏng bồn 4
   AI_TT3219_Bon4_Sim_Pure AT %MD1020 : Real;   // Nhiệt độ mô phỏng chưa có nhiễu bồn 4
   AI_PID_Bon4_Temp_Val_1 AT %MD1024 : Real;   // Biến tạm mô phỏng nhiệt độ 1
   AI_PID_Bon4_Temp_Val_2 AT %MD1028 : Real;   // Biến tạm mô phỏng nhiệt độ 2
   AI_PID_Bon4_Sim_Counter AT %MD1032 : Real;   // Đồng hồ chu kỳ mô phỏng
   AI_PID_Bon4_Sim_Angle AT %MD1036 : Real;   // Góc lượng giác nhiễu
   AI_PID_Bon4_Sim_Sin AT %MD1040 : Real;   // Giá trị hình sin nhiễu
   AI_PID_Bon4_Sim_Noise AT %MD1044 : Real;   // Giá trị nhiễu nhiệt độ
   AI_PLC1_Tip_Bon1_Timer AT %MD1048 : Real;   // Bộ đếm thời gian mô phỏng tip bồn 1
   AI_PLC1_Tip_Bon2_Timer AT %MD1052 : Real;   // Bộ đếm thời gian mô phỏng tip bồn 2
   AI_PLC2_Tip_Bon3_Timer AT %MD1056 : Real;   // Bộ đếm thời gian mô phỏng tip bồn 3
   AI_PLC2_Tip_Bon4_Timer AT %MD1060 : Real;   // Bộ đếm thời gian mô phỏng tip bồn 4
   AI_PID_Bon2_State AT %MW534 : Int;   // Trạng thái khối PID Bồn 2
   AI_PLC1_Stop_Active AT %M339.2 : Bool;   // Tín hiệu dừng active PLC1
   AI_VFD_Bon2_Khuay_Active AT %M339.4 : Bool;   // Trạng thái khuấy Bồn 2 active
   AI_VFD_Bon2_Should_Run AT %M339.5 : Bool;   // Yêu cầu chạy VFD Bồn 2
   AI_HMI_Use_Sim_Input_PLC1 AT %M340.0 : Bool;   // Cho phép sử dụng đầu vào mô phỏng PLC1
   AI_HMI_Use_Sim_Input_BonChua AT %M340.2 : Bool;   // Cho phép sử dụng đầu vào mô phỏng Bồn chứa
   AI_PLC2_Me_Nhanh2_Hoan_Thanh_Nhan_Eff AT %M340.3 : Bool;   // Cờ nhận trạng thái hoàn thành Nhánh 2 hiệu dụng
   AI_PLC2_Me_Nhanh2_Hoan_Thanh_Nhan_HMI_Gated AT %M340.5 : Bool;   // Cờ nhận trạng thái hoàn thành Nhánh 2 HMI gated
   AI_PLC1_SP_Valid AT %M340.7 : Bool;   // Setpoint PLC1 hợp lệ
   AI_BonChua_SP_Valid AT %M341.1 : Bool;   // Setpoint Bồn chứa hợp lệ
   AI_PLC1_Loi_Setpoint AT %M341.2 : Bool;   // Lỗi Setpoint PLC1
   AI_BonChua_Loi_Setpoint AT %M341.4 : Bool;   // Lỗi Setpoint Bồn chứa
   AI_Init_Defaults_Done_PLC1 AT %M341.5 : Bool;   // Khởi tạo Setpoint mặc định PLC1 hoàn tất
   AI_Init_Defaults_Done_BonChua AT %M341.7 : Bool;   // Khởi tạo Setpoint mặc định Bồn chứa hoàn tất
   AI_Init_Trigger_PLC1 AT %M342.0 : Bool;   // Cờ kích hoạt nạp recipe mặc định PLC1
   AI_Init_Trigger_BonChua AT %M342.2 : Bool;   // Cờ kích hoạt nạp recipe mặc định Bồn chứa
   AI_HMI_Load_Default_Recipe AT %M342.3 : Bool;   // Yêu cầu nạp lại Recipe mặc định từ HMI
   AI_PLC1_Load_Default_Cmd AT %M342.4 : Bool;   // Lệnh nạp recipe mặc định gửi sang PLC2
   AI_PLC1_Load_Default_Cmd_M AT %M225.0 : Bool;   // Tag gương phản hồi HMI cho lệnh nạp recipe mặc định PLC1
   AI_PLC1_Load_Default_Done_Nhan AT %M343.1 : Bool;   // Nhận báo nạp recipe xong từ PLC2
   AI_PLC1_Load_Default_Done_Nhan_HMI AT %M111.7 : Bool;   // Tín hiệu mô phỏng/HMI cho nhận báo nạp recipe xong
   AI_PLC1_Load_Default_Done_Nhan_HMI_Gated AT %M343.2 : Bool;   // Tín hiệu nhận báo nạp recipe xong HMI gated
   AI_PLC1_Load_Default_Done_Nhan_Eff AT %M343.3 : Bool;   // Tín hiệu nhận báo nạp recipe xong hiệu dụng
   AI_HMI_Sim_Mode AT %M343.4 : Bool;   // Cho phép toàn bộ tín hiệu mô phỏng HMI tác động vào input hiệu dụng
   AI_HMI_Run_Enable AT %M343.5 : Bool;   // Cho phép vận hành từ HMI ở chế độ thật
   AI_System_Mode_Real AT %M343.6 : Bool;   // Hệ thống đang hoạt động ở chế độ thực tế
   AI_System_Mode_Sim AT %M343.7 : Bool;   // Hệ thống đang hoạt động ở chế độ mô phỏng
   AI_HMI_Sim_Active_Warning AT %M344.0 : Bool;   // Cảnh báo chế độ mô phỏng HMI đang hoạt động
   AI_PID_Bon2_Kp_HMI AT %MD1064 : Real;   // HMI parameter for Kp PID Bồn 2
   AI_PID_Bon2_Ti_HMI AT %MD1068 : Real;   // HMI parameter for Ti PID Bồn 2
   AI_BonChua_Nhan_Dich_Xong_Nhanh1 AT %M344.1 : Bool;   // Nhận dịch xong từ Nhánh 1
   AI_BonChua_Nhan_Dich_Xong_Nhanh2 AT %M344.2 : Bool;   // Nhận dịch xong từ Nhánh 2
   AI_Clock_1Hz_Last AT %M344.3 : Bool;   // Trạng thái Clock 1Hz chu kỳ trước
   AI_Clock_1Hz_Edge AT %M344.4 : Bool;   // Xung cạnh lên của Clock 1Hz
   AI_PLC2_Heartbeat_Last AT %MW540 : Int;   // Heartbeat PLC2 chu kỳ trước
   AI_PLC2_Heartbeat_Changed AT %M344.7 : Bool;   // Cờ heartbeat PLC2 thay đổi
   AI_PLC1_Heartbeat_Timeout AT %M345.0 : Bool;   // Lỗi timeout heartbeat PLC2
   AI_VFD_Bon2_MB_Req AT %M345.1 : Bool;   // REQ cho VFD Modbus
   AI_VFD_Bon2_MB_Mode AT %MB500 : USInt;   // MODE cho VFD Modbus
   AI_VFD_Bon2_MB_DataAddr AT %MD504 : UDInt;   // DATA_ADDR cho VFD Modbus
   AI_VFD_Bon2_MB_DataLen AT %MW508 : UInt;   // DATA_LEN cho VFD Modbus
   AI_VFD_Bon2_MB_DataBuffer AT %MW510 : Word;   // Buffer dữ liệu cho VFD Modbus
END_VAR
